// TIA Portal V16 export
// export: Created 2022-07-21T09:35:16.7270506Z, ExportSetting WithDefaults, DisplayName Totally Integrated Automation Portal, DisplayVersion V16 Update 4, DisplayName TIA Portal Version Control Interface, DisplayVersion V16 Update 2, DisplayName TIA Portal Openness, DisplayVersion V16 Update 4, DisplayName SINAMICS Startdrive Advanced, DisplayVersion V16 Update 5, DisplayName SINAMICS Startdrive G130, G150, S120, S150, SINAMICS MV, S210, DisplayVersion V16 Update 5, DisplayName SINAMICS Startdrive G110M, G120, G120C, G120D, G120P, G115D, DisplayVersion V16 Update 5, DisplayName STEP 7 Professional, DisplayVersion V16 Update 4, DisplayName STEP 7 Safety, DisplayVersion V16, DisplayName WinCC Advanced, DisplayVersion V16 Update 4
FUNCTION_BLOCK "fbIDReadingCognex"   // FB11, LAD
TITLE = Cognex handling / Obsługa kamery Cognex
{ S7_Optimized_Access := 'TRUE' }
VERSION : 0.1
// stored: AutoNumber false, IsIECCheckEnabled true, IsRetainMemResEnabled false, MemoryReserve 100, SetENOAutomatically false, UDAEnableTagReadback false
   VAR_INPUT
      enableDevice { ExternalAccessible := 'False'; ExternalVisible := 'False'; ExternalWritable := 'False'} : Bool;   // Zezwolenie / Enable
      timeBootUp { ExternalAccessible := 'False'; ExternalVisible := 'False'; ExternalWritable := 'False'} : Time := T#5s;   // Czas uruchamiania kamery / Starting time Cognex
      trigger : Bool;   // Wyzwolenie (sekwencja) / Trigger (sequence)
      triggerExtension : Time;   // Wydłużenie sygnału trigger / Extend trigger signal
      timeoutNoData : Time;   // Czas na pobranie danych od zakończenia sygnału trigger / Time for read data since end of trigger signal
      barcodeLength : Int;   // Długość barcode / Barcode length
      resultRightAlligned : Bool;   // Dopasowanie barcode do strony lewa/prawa / Allign barcode left/right
      reTrigger : Bool;   // Aktywacja ponownych odczytów / Activate re-read
      inCamera { ExternalAccessible := 'False'; ExternalVisible := 'False'; ExternalWritable := 'False'} : "typeIDReadingInputsCognex";   // Wejścia z kamery Cognex / Inputs from Cognex
      group : "typeGroup";   // Grupa / Group
   END_VAR
   VAR_OUTPUT
      outCamera { ExternalAccessible := 'False'; ExternalVisible := 'False'; ExternalWritable := 'False'} : "typeIDReadingOutputsCognex";   // Wyjścia do kamery Cognex / Outputs to Cognex
   END_VAR
   VAR_IN_OUT
      data : "typeCognex";   // Dane HMI cognex / HMI Cognex data
   END_VAR
   VAR
      instGetInstancePath { ExternalAccessible := 'False'; ExternalVisible := 'False'; ExternalWritable := 'False'; S7_SetPoint := 'True'} : "fbGetInstancePath";
      instReadingWindow : "fbReadingWindow";
      sInstancePath { ExternalAccessible := 'False'; ExternalVisible := 'False'; ExternalWritable := 'False'} : String[100];
      statMemREResultAvailable { ExternalAccessible := 'False'; ExternalVisible := 'False'; ExternalWritable := 'False'} : Bool;   // Rezultat dostępny flaga pomocnicza / Result available temporary bit
      statREWaitingForData : Bool;   // Zbocze narastające / Positive edge
      statFEWaitingData { S7_SetPoint := 'True'} : Bool;   // Zbocze opadające / Negative edge
      statAmountofChars { ExternalAccessible := 'False'; ExternalVisible := 'False'; ExternalWritable := 'False'} : UInt;   // Liczba odczytanych znaków / Amount of read characters
      instMessageErrorDevice { ExternalAccessible := 'False'; ExternalVisible := 'False'; ExternalWritable := 'False'; S7_SetPoint := 'True'} : "fbMessageError";
      instMessageRate { ExternalAccessible := 'False'; ExternalVisible := 'False'; ExternalWritable := 'False'; S7_SetPoint := 'True'} : "fbMessageHandlingRate";
      instMessageTrigger { ExternalAccessible := 'False'; ExternalVisible := 'False'; ExternalWritable := 'False'; S7_SetPoint := 'True'} : "fbMessageHandlingRate";
      instRestTimeTrigger { S7_SetPoint := 'True'} : TP_TIME;
      instTOnBootUpDevice { ExternalAccessible := 'False'; ExternalVisible := 'False'; ExternalWritable := 'False'; S7_SetPoint := 'True'} : TON_TIME;
      instTOnRstError { ExternalAccessible := 'False'; ExternalVisible := 'False'; ExternalWritable := 'False'; S7_SetPoint := 'True'} : TON_TIME;
      sBootUpCompleteDevice { ExternalAccessible := 'False'; ExternalVisible := 'False'; ExternalWritable := 'False'} : Bool;
      sMonitoring : Struct
         TriggerCount1 : Int;
         TriggerCount2 : Int;
      END_STRUCT;
   END_VAR
   VAR_TEMP
      tExpextedData : Bool;
      tDiff : Int;
      tAddString : String;
      tEnableDeviceMessages : Bool;
      tTrigger : Bool;
      tMsgError : Bool;
      tNoDataEdge : Bool;
      tAmountTillMsg : USInt;
   END_VAR
   VAR CONSTANT
      constFiller : Char := '_';
      constNoRead : Char := '?';
      constInvalidData : Char := '!';
      constNoData : Char := '0';
      constRateWarning : Real := 100.0;
      constRateError : Real := 100.0;
      constCountTillMessage : USInt := 1;
   END_VAR
   VAR_TEMP   // added for the SCL form of the ladder/FBD networks
      _w1 : Bool;
   END_VAR
BEGIN

REGION Network 1: Trigger / Wyzwolenie
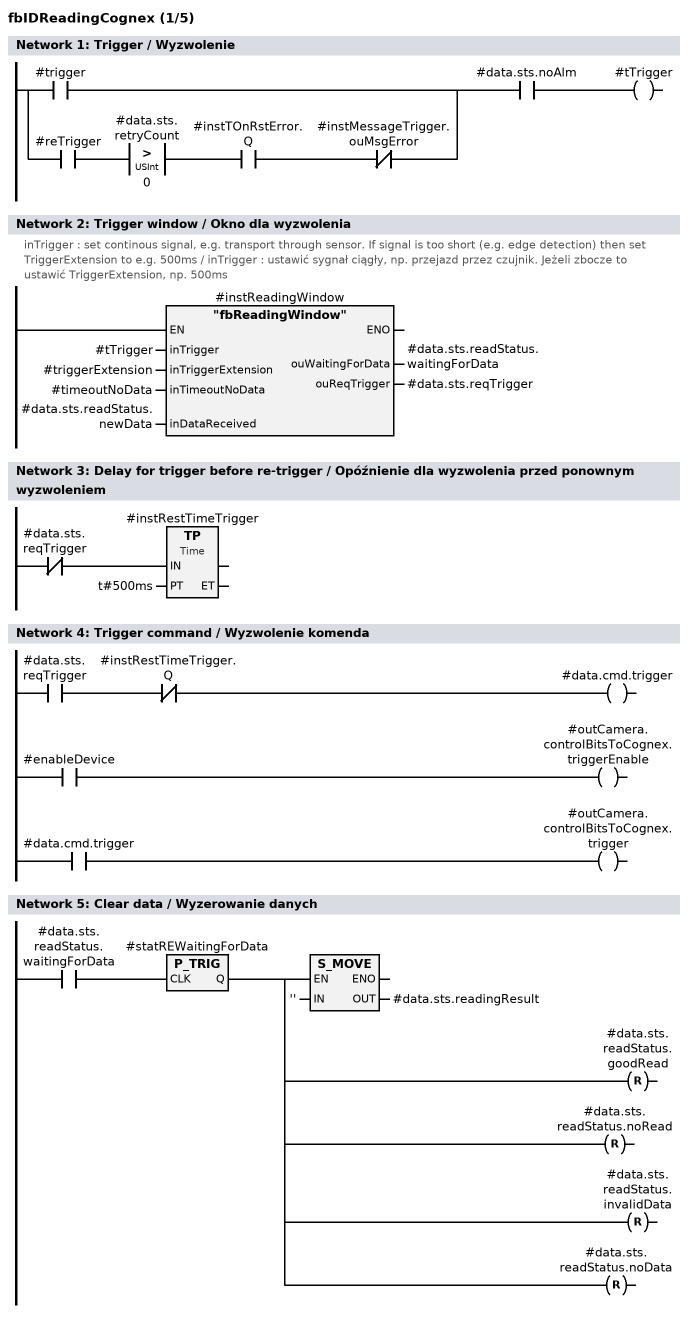
   RUNG wire#powerrail
      Contact( #trigger )
      wire#w1
      Contact( #data.sts.noAlm )
      Coil( #tTrigger )
   END_RUNG
   RUNG wire#powerrail
      Contact( #reTrigger )
      { S7_Templates := "SrcType := USInt" } GT_Contact(in1 := #data.sts.retryCount, in2 := 0)
      Contact( #instTOnRstError.Q )
      I_Contact( #instMessageTrigger.ouMsgError )
   END_RUNG wire#w1
   // the same network as SCL:
   #tTrigger := (#trigger OR (#reTrigger AND (#data.sts.retryCount > 0) AND #instTOnRstError.Q AND NOT #instMessageTrigger.ouMsgError)) AND #data.sts.noAlm;
END_REGION

REGION Network 2: Trigger window / Okno dla wyzwolenia
   // inTrigger : set continous signal, e.g. transport through sensor. If signal is too short (e.g. edge detection) then set TriggerExtension to e.g. 500ms / inTrigger : ustawić sygnał ciągły, np. przejazd przez czujnik. Jeżeli zbocze to ustawić TriggerExtension, np. 500ms
   RUNG wire#powerrail
      #instReadingWindow(inTrigger := #tTrigger, inTriggerExtension := #triggerExtension, inTimeoutNoData := #timeoutNoData, inDataReceived := #data.sts.readStatus.newData, ouWaitingForData => #data.sts.readStatus.waitingForData, ouReqTrigger => #data.sts.reqTrigger)
   END_RUNG
   // the same network as SCL:
   #instReadingWindow(inTrigger := #tTrigger,   // "fbReadingWindow"
                      inTriggerExtension := #triggerExtension,
                      inTimeoutNoData := #timeoutNoData,
                      inDataReceived := #data.sts.readStatus.newData,
                      ouWaitingForData => #data.sts.readStatus.waitingForData,
                      ouReqTrigger => #data.sts.reqTrigger);
END_REGION

REGION Network 3: Delay for trigger before re-trigger / Opóźnienie dla wyzwolenia przed ponownym wyzwoleniem
   RUNG wire#powerrail
      I_Contact( #data.sts.reqTrigger )
      { S7_Templates := "time_type := Time" } #instRestTimeTrigger.TP(pt := t#500ms, et =>)
   END_RUNG
   // the same network as SCL:
   #instRestTimeTrigger(IN := NOT #data.sts.reqTrigger, PT := t#500ms);   // TP
END_REGION

REGION Network 4: Trigger command / Wyzwolenie komenda
   RUNG wire#powerrail
      Contact( #data.sts.reqTrigger )
      I_Contact( #instRestTimeTrigger.Q )
      Coil( #data.cmd.trigger )
   END_RUNG
   RUNG wire#powerrail
      Contact( #enableDevice )
      Coil( #outCamera.controlBitsToCognex.triggerEnable )
   END_RUNG
   RUNG wire#powerrail
      Contact( #data.cmd.trigger )
      Coil( #outCamera.controlBitsToCognex.trigger )
   END_RUNG
   // the same network as SCL:
   #data.cmd.trigger := #data.sts.reqTrigger AND NOT #instRestTimeTrigger.Q;
   #outCamera.controlBitsToCognex.triggerEnable := #enableDevice;
   #outCamera.controlBitsToCognex.trigger := #data.cmd.trigger;
END_REGION

REGION Network 5: Clear data / Wyzerowanie danych
   RUNG wire#powerrail
      Contact( #data.sts.readStatus.waitingForData )
      P_Trig( #statREWaitingForData )
      wire#w1
      { S7_GenerateENO := "TRUE" } S_Move(in := '', out => #data.sts.readingResult)
   END_RUNG
   RUNG wire#w1
      R_Coil( #data.sts.readStatus.goodRead )
   END_RUNG
   RUNG wire#w1
      R_Coil( #data.sts.readStatus.noRead )
   END_RUNG
   RUNG wire#w1
      R_Coil( #data.sts.readStatus.invalidData )
   END_RUNG
   RUNG wire#w1
      R_Coil( #data.sts.readStatus.noData )
   END_RUNG
   // the same network as SCL:
   #_w1 := #data.sts.readStatus.waitingForData AND NOT #statREWaitingForData;   // rising edge
   #statREWaitingForData := #data.sts.readStatus.waitingForData;
   IF #_w1 THEN
       #data.sts.readingResult := '';
       #data.sts.readStatus.goodRead := FALSE;
       #data.sts.readStatus.noRead := FALSE;
       #data.sts.readStatus.invalidData := FALSE;
       #data.sts.readStatus.noData := FALSE;
   END_IF;
END_REGION

REGION Network 6: No data / Brak danych
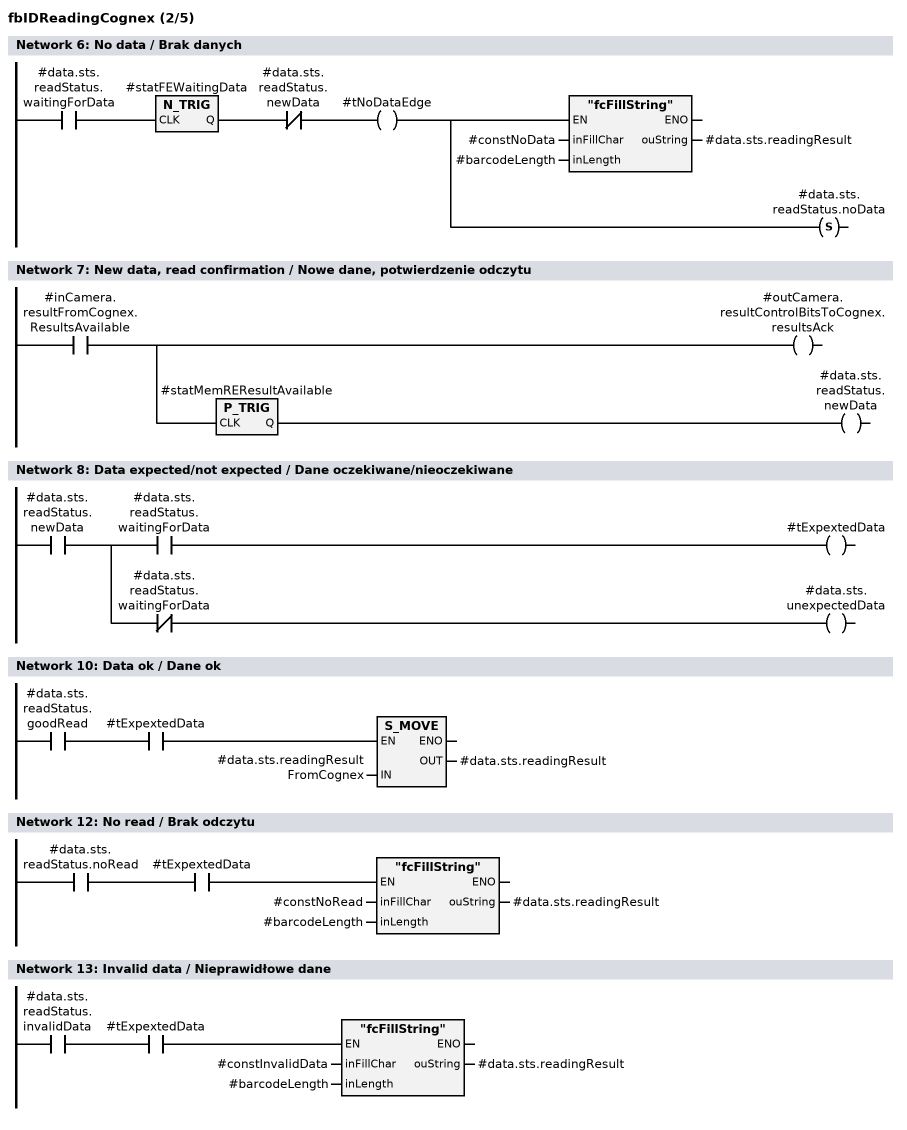
   RUNG wire#powerrail
      Contact( #data.sts.readStatus.waitingForData )
      N_Trig( #statFEWaitingData )
      I_Contact( #data.sts.readStatus.newData )
      Coil( #tNoDataEdge )
      wire#w1
      "fcFillString"(inFillChar := #constNoData, inLength := #barcodeLength, ouString => #data.sts.readingResult)
   END_RUNG
   RUNG wire#w1
      S_Coil( #data.sts.readStatus.noData )
   END_RUNG
   // the same network as SCL:
   #_w1 := NOT #data.sts.readStatus.waitingForData AND #statFEWaitingData;   // falling edge
   #statFEWaitingData := #data.sts.readStatus.waitingForData;
   #tNoDataEdge := #_w1 AND NOT #data.sts.readStatus.newData;
   IF #tNoDataEdge THEN
       "fcFillString"(inFillChar := #constNoData, inLength := #barcodeLength, ouString => #data.sts.readingResult);
       #data.sts.readStatus.noData := TRUE;
   END_IF;
END_REGION

REGION Network 7: New data, read confirmation / Nowe dane, potwierdzenie odczytu
   RUNG wire#powerrail
      Contact( #inCamera.resultFromCognex.ResultsAvailable )
      wire#w1
      Coil( #outCamera.resultControlBitsToCognex.resultsAck )
   END_RUNG
   RUNG wire#w1
      P_Trig( #statMemREResultAvailable )
      Coil( #data.sts.readStatus.newData )
   END_RUNG
   // the same network as SCL:
   #outCamera.resultControlBitsToCognex.resultsAck := #inCamera.resultFromCognex.ResultsAvailable;
   #_w1 := #inCamera.resultFromCognex.ResultsAvailable AND NOT #statMemREResultAvailable;   // rising edge
   #statMemREResultAvailable := #inCamera.resultFromCognex.ResultsAvailable;
   #data.sts.readStatus.newData := #_w1;
END_REGION

REGION Network 8: Data expected/not expected / Dane oczekiwane/nieoczekiwane
   RUNG wire#powerrail
      Contact( #data.sts.readStatus.newData )
      wire#w1
      Contact( #data.sts.readStatus.waitingForData )
      Coil( #tExpextedData )
   END_RUNG
   RUNG wire#w1
      I_Contact( #data.sts.readStatus.waitingForData )
      Coil( #data.sts.unexpectedData )
   END_RUNG
   // the same network as SCL:
   #tExpextedData := #data.sts.readStatus.newData AND #data.sts.readStatus.waitingForData;
   #data.sts.unexpectedData := #data.sts.readStatus.newData AND NOT #data.sts.readStatus.waitingForData;
END_REGION

REGION Network 9 (SCL): New data - before processing / Nowe dane - do obróbki

   // setting for readStatus and readingResultFromCognex (no output yet, only to evaluate !)
   IF #data.sts.readStatus.newData THEN

       #data.sts.readStatus.goodRead := FALSE;
       #data.sts.readStatus.noRead := FALSE;
       #data.sts.readStatus.invalidData := FALSE;

       #statAmountofChars := WORD_TO_UINT(#inCamera.resultDataFromCognex.ResultLength);

       // Get reading status
       IF #inCamera.resultDataFromCognex.GoodRead THEN
           REGION Good Read            
               #data.sts.readStatus.goodRead := TRUE;
               // Copy barcode
               Chars_TO_Strg(Chars := #inCamera.resultDataFromCognex.inspectionResults,
                             pChars := 0,
                             Cnt := #statAmountofChars,
                             Strg => #data.sts.readingResultFromCognex);
           END_REGION
       ELSIF NOT #inCamera.resultFromCognex.GeneralFault THEN
           REGION No Read
               #data.sts.readStatus.noRead := TRUE;
               #data.sts.readingResultFromCognex := '';
           END_REGION
       ELSE
           REGION Invalid Data
               #data.sts.readStatus.invalidData := TRUE;
               // Copy barcode
               Chars_TO_Strg(Chars := #inCamera.resultDataFromCognex.inspectionResults,
                             pChars := 0,
                             Cnt := #statAmountofChars,
                             Strg => #data.sts.readingResultFromCognex);

           END_REGION
       END_IF;
   END_IF;
END_REGION

REGION Network 10: Data ok / Dane ok
   RUNG wire#powerrail
      Contact( #data.sts.readStatus.goodRead )
      Contact( #tExpextedData )
      { S7_GenerateENO := "TRUE" } S_Move(in := #data.sts.readingResultFromCognex, out => #data.sts.readingResult)
   END_RUNG
   // the same network as SCL:
   IF #data.sts.readStatus.goodRead AND #tExpextedData THEN
       #data.sts.readingResult := #data.sts.readingResultFromCognex;
   END_IF;
END_REGION

REGION Network 11 (SCL): Data ok - supplement information / Dane ok - uzupełnienie informacji

   //max length - max string length 
   #tDiff := #barcodeLength - LEN(#data.sts.readingResult);

   // check if reading result is long enough
   IF #tDiff <> 0 AND #data.sts.readStatus.goodRead THEN
     // build string to add to reading result
     #tAddString := '';
     FOR #tDiff := #tDiff TO 1 BY -1 DO
         #tAddString := CONCAT(IN1 := #tAddString, IN2 := #constFiller);
     END_FOR;
     // add string to reading result either as prefix or suffix
     IF #resultRightAlligned THEN
         #data.sts.readingResult := CONCAT(IN1:=#tAddString,IN2:=#data.sts.readingResult);
     ELSE
         #data.sts.readingResult := CONCAT(IN1:=#data.sts.readingResult,IN2:=#tAddString);
     END_IF;
   END_IF;
END_REGION

REGION Network 12: No read / Brak odczytu
   RUNG wire#powerrail
      Contact( #data.sts.readStatus.noRead )
      Contact( #tExpextedData )
      "fcFillString"(inFillChar := #constNoRead, inLength := #barcodeLength, ouString => #data.sts.readingResult)
   END_RUNG
   // the same network as SCL:
   IF #data.sts.readStatus.noRead AND #tExpextedData THEN
       "fcFillString"(inFillChar := #constNoRead, inLength := #barcodeLength, ouString => #data.sts.readingResult);
   END_IF;
END_REGION

REGION Network 13: Invalid data / Nieprawidłowe dane
   RUNG wire#powerrail
      Contact( #data.sts.readStatus.invalidData )
      Contact( #tExpextedData )
      "fcFillString"(inFillChar := #constInvalidData, inLength := #barcodeLength, ouString => #data.sts.readingResult)
   END_RUNG
   // the same network as SCL:
   IF #data.sts.readStatus.invalidData AND #tExpextedData THEN
       "fcFillString"(inFillChar := #constInvalidData,
                      inLength := #barcodeLength,
                      ouString => #data.sts.readingResult);
   END_IF;
END_REGION

REGION Network 14: Error handling / Obsługa błędów
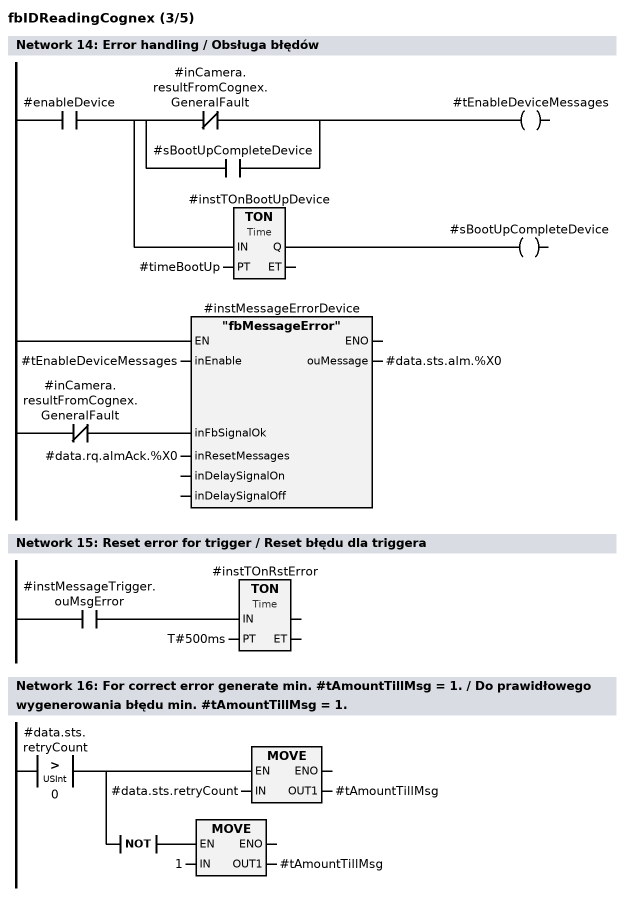
   RUNG wire#powerrail
      Contact( #enableDevice )
      wire#w1
      I_Contact( #inCamera.resultFromCognex.GeneralFault )
      wire#w2
      Coil( #tEnableDeviceMessages )
   END_RUNG
   RUNG wire#w1
      Contact( #sBootUpCompleteDevice )
   END_RUNG wire#w2
   RUNG wire#w1
      { S7_Templates := "time_type := Time" } #instTOnBootUpDevice.TON(pt := #timeBootUp, et =>)
      Coil( #sBootUpCompleteDevice )
   END_RUNG
   RUNG wire#powerrail
      #instMessageErrorDevice(inFbSignalOk := wire#w3, inEnable := #tEnableDeviceMessages, inResetMessages := #data.rq.almAck.%X0, inDelaySignalOn :=, inDelaySignalOff :=, ouMessage => #data.sts.alm.%X0)
   END_RUNG
   RUNG wire#powerrail
      I_Contact( #inCamera.resultFromCognex.GeneralFault )
   END_RUNG wire#w3
   // the same network as SCL:
   #tEnableDeviceMessages := #enableDevice AND (NOT #inCamera.resultFromCognex.GeneralFault OR #sBootUpCompleteDevice);
   #instTOnBootUpDevice(IN := #enableDevice, PT := #timeBootUp);   // TON
   #sBootUpCompleteDevice := #instTOnBootUpDevice.Q;
   #instMessageErrorDevice(inEnable := #tEnableDeviceMessages,   // "fbMessageError"
                           inFbSignalOk := NOT #inCamera.resultFromCognex.GeneralFault,
                           inResetMessages := #data.rq.almAck.%X0,
                           ouMessage => #data.sts.alm.%X0);
END_REGION

REGION Network 15: Reset error for trigger / Reset błędu dla triggera
   RUNG wire#powerrail
      Contact( #instMessageTrigger.ouMsgError )
      { S7_Templates := "time_type := Time" } #instTOnRstError.TON(pt := T#500ms, et =>)
   END_RUNG
   // the same network as SCL:
   #instTOnRstError(IN := #instMessageTrigger.ouMsgError, PT := T#500ms);   // TON
END_REGION

REGION Network 16: For correct error generate min. #tAmountTillMsg = 1. / Do prawidłowego wygenerowania błędu min. #tAmountTillMsg = 1.
   RUNG wire#powerrail
      { S7_Templates := "SrcType := USInt" } GT_Contact(in1 := #data.sts.retryCount, in2 := 0)
      wire#w1
      Move(in := #data.sts.retryCount, out1 => #tAmountTillMsg)
   END_RUNG
   RUNG wire#w1
      Not()
      Move(in := 1, out1 => #tAmountTillMsg)
   END_RUNG
   // the same network as SCL:
   #_w1 := #data.sts.retryCount > 0;
   IF #_w1 THEN #tAmountTillMsg := #data.sts.retryCount; END_IF;
   IF NOT #_w1 THEN #tAmountTillMsg := 1; END_IF;
END_REGION

REGION Network 17: Re-trigger / Ponowne wyzwolenie kamery
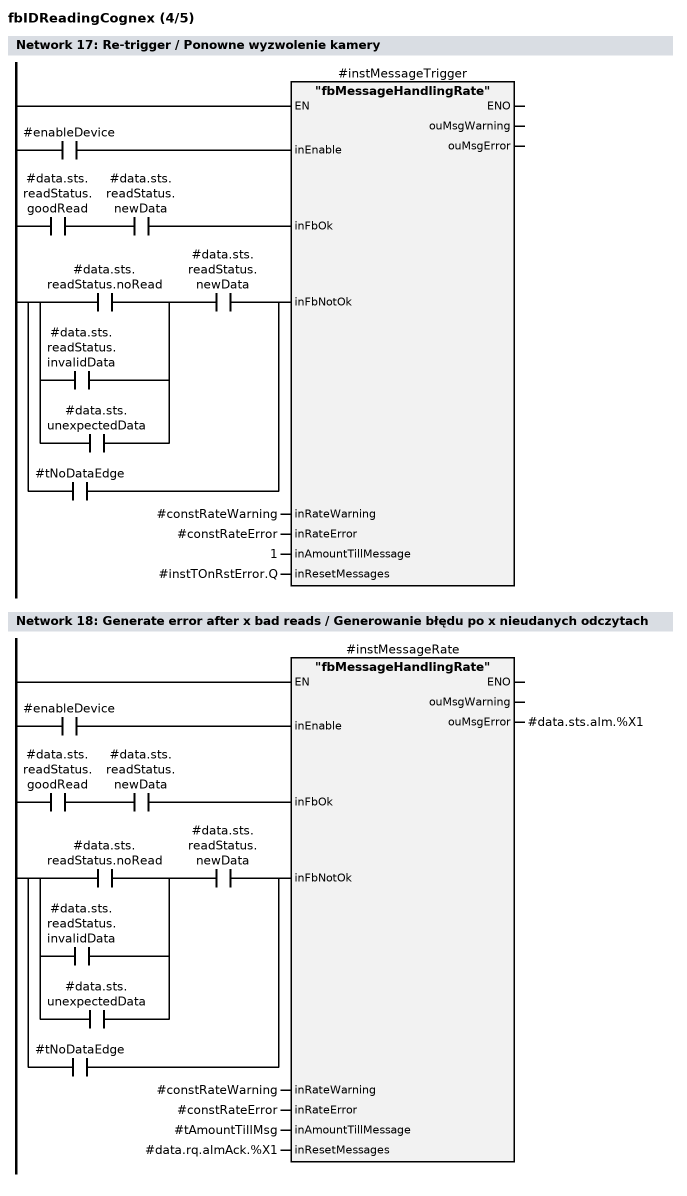
   RUNG wire#powerrail
      #instMessageTrigger(inEnable := wire#w1, inFbOk := wire#w2, inFbNotOk := wire#w4, inRateWarning := #constRateWarning, inRateError := #constRateError, inAmountTillMessage := 1, inResetMessages := #instTOnRstError.Q, ouMsgWarning =>, ouMsgError =>)
   END_RUNG
   RUNG wire#powerrail
      Contact( #enableDevice )
   END_RUNG wire#w1
   RUNG wire#powerrail
      Contact( #data.sts.readStatus.goodRead )
      Contact( #data.sts.readStatus.newData )
   END_RUNG wire#w2
   RUNG wire#powerrail
      Contact( #data.sts.readStatus.noRead )
      wire#w3
      Contact( #data.sts.readStatus.newData )
   END_RUNG wire#w4
   RUNG wire#powerrail
      Contact( #data.sts.readStatus.invalidData )
   END_RUNG wire#w3
   RUNG wire#powerrail
      Contact( #data.sts.unexpectedData )
   END_RUNG wire#w3
   RUNG wire#powerrail
      Contact( #tNoDataEdge )
   END_RUNG wire#w4
   // the same network as SCL:
   #instMessageTrigger(inEnable := #enableDevice,   // "fbMessageHandlingRate"
                       inFbOk := #data.sts.readStatus.goodRead AND #data.sts.readStatus.newData,
                       inFbNotOk := ((#data.sts.readStatus.noRead OR #data.sts.readStatus.invalidData OR #data.sts.unexpectedData) AND #data.sts.readStatus.newData) OR #tNoDataEdge,
                       inRateWarning := #constRateWarning,
                       inRateError := #constRateError,
                       inAmountTillMessage := 1,
                       inResetMessages := #instTOnRstError.Q);
END_REGION

REGION Network 18: Generate error after x bad reads / Generowanie błędu po x nieudanych odczytach
   RUNG wire#powerrail
      #instMessageRate(inEnable := wire#w1, inFbOk := wire#w2, inFbNotOk := wire#w4, inRateWarning := #constRateWarning, inRateError := #constRateError, inAmountTillMessage := #tAmountTillMsg, inResetMessages := #data.rq.almAck.%X1, ouMsgWarning =>, ouMsgError => #data.sts.alm.%X1)
   END_RUNG
   RUNG wire#powerrail
      Contact( #enableDevice )
   END_RUNG wire#w1
   RUNG wire#powerrail
      Contact( #data.sts.readStatus.goodRead )
      Contact( #data.sts.readStatus.newData )
   END_RUNG wire#w2
   RUNG wire#powerrail
      Contact( #data.sts.readStatus.noRead )
      wire#w3
      Contact( #data.sts.readStatus.newData )
   END_RUNG wire#w4
   RUNG wire#powerrail
      Contact( #data.sts.readStatus.invalidData )
   END_RUNG wire#w3
   RUNG wire#powerrail
      Contact( #data.sts.unexpectedData )
   END_RUNG wire#w3
   RUNG wire#powerrail
      Contact( #tNoDataEdge )
   END_RUNG wire#w4
   // the same network as SCL:
   #instMessageRate(inEnable := #enableDevice,   // "fbMessageHandlingRate"
                    inFbOk := #data.sts.readStatus.goodRead AND #data.sts.readStatus.newData,
                    inFbNotOk := ((#data.sts.readStatus.noRead OR #data.sts.readStatus.invalidData OR #data.sts.unexpectedData) AND #data.sts.readStatus.newData) OR #tNoDataEdge,
                    inRateWarning := #constRateWarning,
                    inRateError := #constRateError,
                    inAmountTillMessage := #tAmountTillMsg,
                    inResetMessages := #data.rq.almAck.%X1,
                    ouMsgError => #data.sts.alm.%X1);
END_REGION

REGION Network 19 (SCL): Akceptuj numer LOT użytkownika
   IF #data.rq.acceptUserLOT THEN
       #data.sts.readingResult := #data.rq.userLOT;
   END_IF;
END_REGION

REGION Network 20: Outputs / Wyjścia
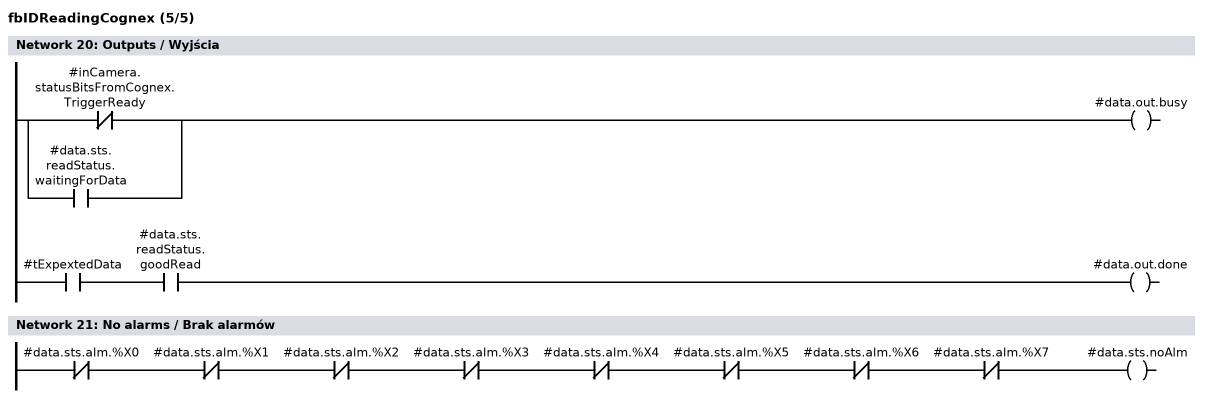
   RUNG wire#powerrail
      I_Contact( #inCamera.statusBitsFromCognex.TriggerReady )
      wire#w1
      Coil( #data.out.busy )
   END_RUNG
   RUNG wire#powerrail
      Contact( #data.sts.readStatus.waitingForData )
   END_RUNG wire#w1
   RUNG wire#powerrail
      Contact( #tExpextedData )
      Contact( #data.sts.readStatus.goodRead )
      Coil( #data.out.done )
   END_RUNG
   // the same network as SCL:
   #data.out.busy := NOT #inCamera.statusBitsFromCognex.TriggerReady OR #data.sts.readStatus.waitingForData;
   #data.out.done := #tExpextedData AND #data.sts.readStatus.goodRead;
END_REGION

REGION Network 21: No alarms / Brak alarmów
   RUNG wire#powerrail
      I_Contact( #data.sts.alm.%X0 )
      I_Contact( #data.sts.alm.%X1 )
      I_Contact( #data.sts.alm.%X2 )
      I_Contact( #data.sts.alm.%X3 )
      I_Contact( #data.sts.alm.%X4 )
      I_Contact( #data.sts.alm.%X5 )
      I_Contact( #data.sts.alm.%X6 )
      I_Contact( #data.sts.alm.%X7 )
      Coil( #data.sts.noAlm )
   END_RUNG
   // the same network as SCL:
   #data.sts.noAlm := NOT #data.sts.alm.%X0 AND NOT #data.sts.alm.%X1 AND NOT #data.sts.alm.%X2 AND NOT #data.sts.alm.%X3 AND NOT #data.sts.alm.%X4 AND NOT #data.sts.alm.%X5 AND NOT #data.sts.alm.%X6 AND NOT #data.sts.alm.%X7;
END_REGION
END_FUNCTION_BLOCK
